INTERFACE IEventLogger

METHOD LogEvent : bool
VAR_INPUT
	sMessage : STRING;
END_VAR
END_METHOD

END_INTERFACE

(* stored: Version 1.1.0.1
   Itf IEventLogger: Id {db077830-80db-4e14-bad0-faab95f85615}
   Method LogEvent: Id {b4fe520d-5c5b-4e87-a92b-807a4236d043} *)
